// TIA Portal V16 export
// export: Created 2021-11-15T19:59:24.1502898Z, ExportSetting WithDefaults, DisplayName Totally Integrated Automation Portal, DisplayVersion V16, DisplayName TIA Portal Version Control Interface, DisplayVersion V16, DisplayName TIA Portal Openness, DisplayVersion V16, DisplayName TIA Portal Teamcenter Gateway, DisplayVersion V16, DisplayName STEP 7 Professional, DisplayVersion V16, DisplayName STEP 7 Safety, DisplayVersion V16, DisplayName WinCC Professional, DisplayVersion V16
ORGANIZATION_BLOCK "Main"   // OB1, LAD, ProgramCycle
TITLE = "Main Program Sweep (Cycle)"
{ S7_Optimized_Access := 'TRUE' }
VERSION : 0.1
// stored: AutoNumber true, IsIECCheckEnabled false, SetENOAutomatically false
BEGIN

REGION Network 1
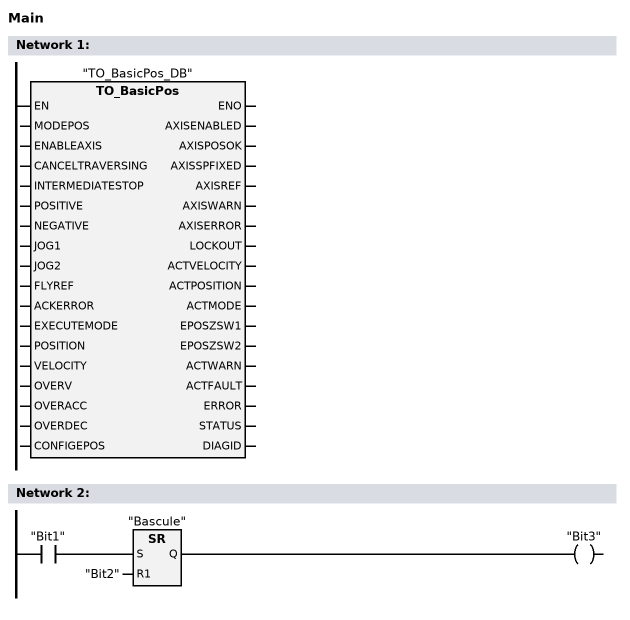
   RUNG wire#powerrail
      "TO_BasicPos_DB".TO_BasicPos(ModePos :=, EnableAxis :=, CancelTraversing :=, IntermediateStop :=, Positive :=, Negative :=, Jog1 :=, Jog2 :=, FlyRef :=, AckError :=, ExecuteMode :=, Position :=, Velocity :=, OverV :=, OverAcc :=, OverDec :=, ConfigEPos :=, AxisEnabled =>, AxisPosOk =>, AxisSpFixed =>, AxisRef =>, AxisWarn =>, AxisError =>, Lockout =>, ActVelocity =>, ActPosition =>, ActMode =>, EPosZSW1 =>, EPosZSW2 =>, ActWarn =>, ActFault =>, Error =>, Status =>, DiagId =>)
   END_RUNG
   // the same network as SCL:
   "TO_BasicPos_DB"();   // TO_BasicPos
END_REGION

REGION Network 2
   RUNG wire#powerrail
      Contact( "Bit1" )
      S_SR(operand := "Bascule", r1 := "Bit2")
      Coil( "Bit3" )
   END_RUNG
   // the same network as SCL:
   IF "Bit1" THEN
       "Bascule" := TRUE;   // SR flip-flop
   END_IF;
   IF "Bit2" THEN "Bascule" := FALSE; END_IF;
   "Bit3" := "Bascule";
END_REGION
END_ORGANIZATION_BLOCK
